(* CODESYS project MakeBagSequence.xml

Project tree, tasks and I/O mapping:
  function block MakeBagSequence [SFC]
*)

// MakeBagSequence
FUNCTION_BLOCK MakeBagSequence
VAR_INPUT
	SFCInit: BOOL;
	Trigger: BOOL;
	BagReady: BOOL;
	BagOpenFailed: BOOL;
	IceFilled: BOOL;
	HeatSealClosed: BOOL;
	BagSealed: BOOL;
END_VAR
VAR_OUTPUT
	BlowerOn: BOOL;
	AdvanceBag: BOOL;
	FillIce: BOOL;
	SealBag: BOOL;
	TearBag: BOOL;
	PresentBag: BOOL;
END_VAR
VAR
END_VAR

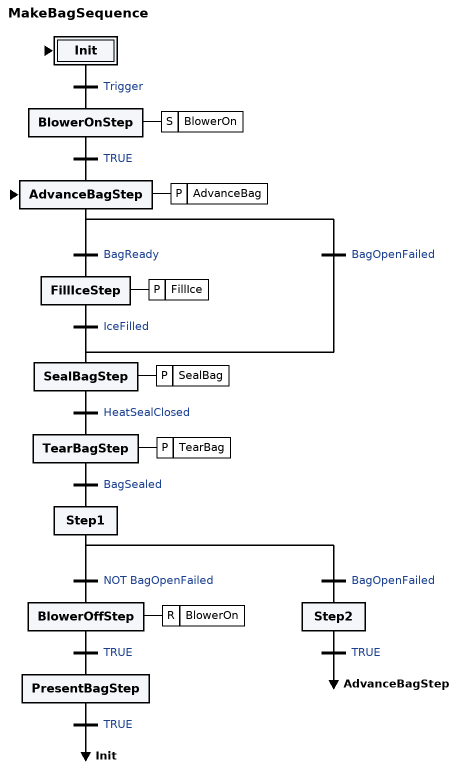
INITIAL_STEP Init:
END_STEP
TRANSITION FROM Init TO BlowerOnStep
    := Trigger;
END_TRANSITION
STEP BlowerOnStep:
    BlowerOn(S);
END_STEP
TRANSITION FROM BlowerOnStep TO AdvanceBagStep
    := TRUE;
END_TRANSITION
STEP AdvanceBagStep:
    AdvanceBag(P);
END_STEP
TRANSITION FROM AdvanceBagStep TO FillIceStep
    := BagReady;
END_TRANSITION
STEP FillIceStep:
    FillIce(P);
END_STEP
TRANSITION FROM FillIceStep TO SealBagStep
    := IceFilled;
END_TRANSITION
TRANSITION FROM AdvanceBagStep TO SealBagStep
    := BagOpenFailed;
END_TRANSITION
STEP SealBagStep:
    SealBag(P);
END_STEP
TRANSITION FROM SealBagStep TO TearBagStep
    := HeatSealClosed;
END_TRANSITION
STEP TearBagStep:
    TearBag(P);
END_STEP
TRANSITION FROM TearBagStep TO Step1
    := BagSealed;
END_TRANSITION
STEP Step1:
END_STEP
TRANSITION FROM Step1 TO BlowerOffStep
    := NOT BagOpenFailed;
END_TRANSITION
TRANSITION FROM Step1 TO Step2
    := BagOpenFailed;
END_TRANSITION
STEP Step2:
END_STEP
TRANSITION FROM Step2 TO AdvanceBagStep
    := TRUE;
END_TRANSITION
STEP BlowerOffStep:
    BlowerOn(R);
END_STEP
TRANSITION FROM BlowerOffStep TO PresentBagStep
    := TRUE;
END_TRANSITION
STEP PresentBagStep:
END_STEP
TRANSITION FROM PresentBagStep TO Init
    := TRUE;
END_TRANSITION

END_FUNCTION_BLOCK
